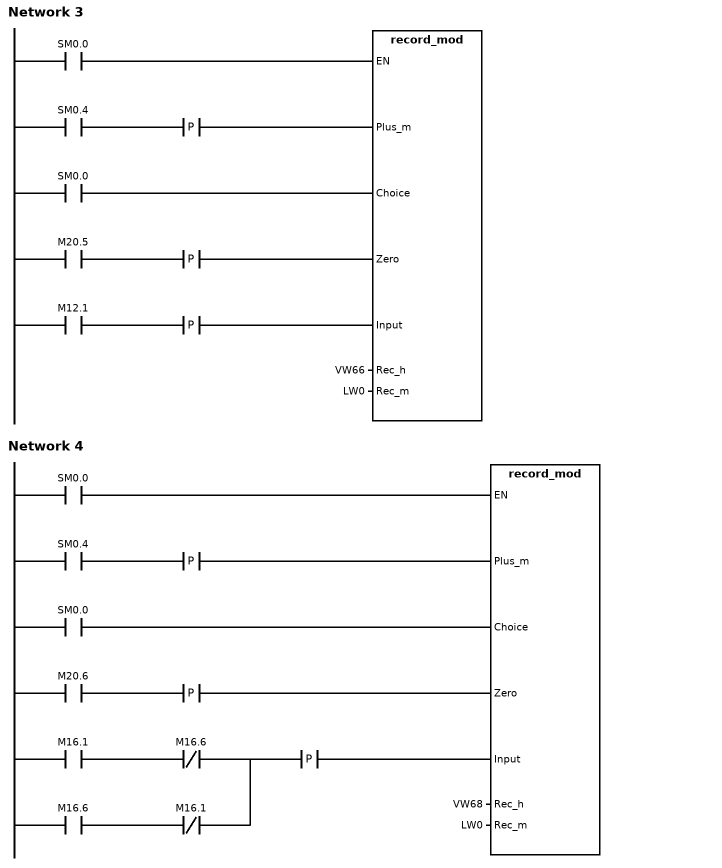
[picture p24: SBR11 networks 3-4]
Network 3
LD     SM0.0
=      L60.0
LD     SM0.4
EU
=      L63.7
LD     SM0.0
=      L63.6
LD     M20.5
EU
=      L63.5
LD     M12.1
EU
=      L63.4
LD     L60.0
CALL   record_mod:SBR13, L63.7, L63.6, L63.5, L63.4, VW66, LW0
Network 4
LD     SM0.0
=      L60.0
LD     SM0.4
EU
=      L63.7
LD     SM0.0
=      L63.6
LD     M20.6
EU
=      L63.5
LD     M16.1
AN     M16.6
LD     M16.6
AN     M16.1
OLD
EU
=      L63.4
LD     L60.0
CALL   record_mod:SBR13, L63.7, L63.6, L63.5, L63.4, VW68, LW0
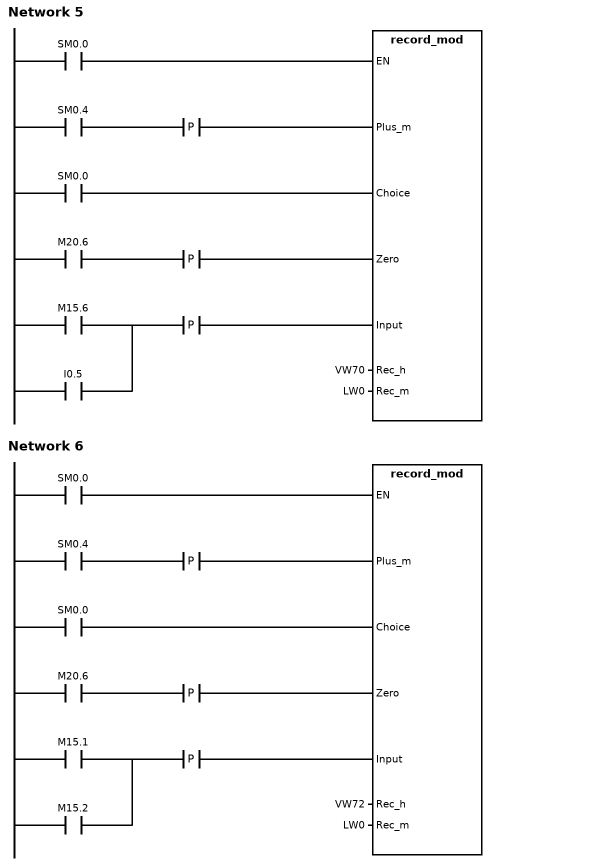
Network 5
LD     SM0.0
=      L60.0
LD     SM0.4
EU
=      L63.7
LD     SM0.0
=      L63.6
LD     M20.6
EU
=      L63.5
LD     M15.6
O      I0.5
EU
=      L63.4
LD     L60.0
CALL   record_mod:SBR13, L63.7, L63.6, L63.5, L63.4, VW70, LW0
Network 6
LD     SM0.0
=      L60.0
LD     SM0.4
EU
=      L63.7
LD     SM0.0
=      L63.6
LD     M20.6
EU
=      L63.5
LD     M15.1
O      M15.2
EU
=      L63.4
LD     L60.0
CALL   record_mod:SBR13, L63.7, L63.6, L63.5, L63.4, VW72, LW0
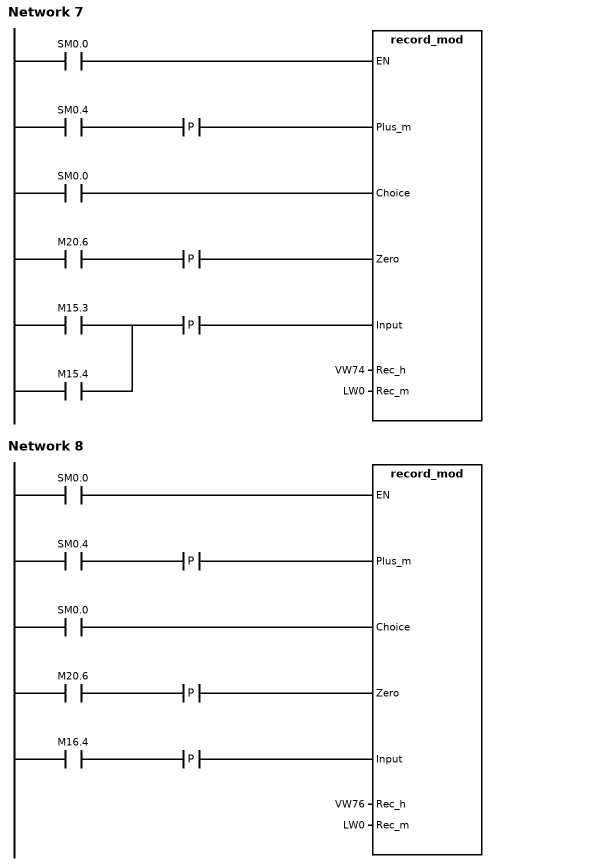
Network 7
LD     SM0.0
=      L60.0
LD     SM0.4
EU
=      L63.7
LD     SM0.0
=      L63.6
LD     M20.6
EU
=      L63.5
LD     M15.3
O      M15.4
EU
=      L63.4
LD     L60.0
CALL   record_mod:SBR13, L63.7, L63.6, L63.5, L63.4, VW74, LW0
Network 8
LD     SM0.0
=      L60.0
LD     SM0.4
EU
=      L63.7
LD     SM0.0
=      L63.6
LD     M20.6
EU
=      L63.5
LD     M16.4
EU
=      L63.4
LD     L60.0
CALL   record_mod:SBR13, L63.7, L63.6, L63.5, L63.4, VW76, LW0
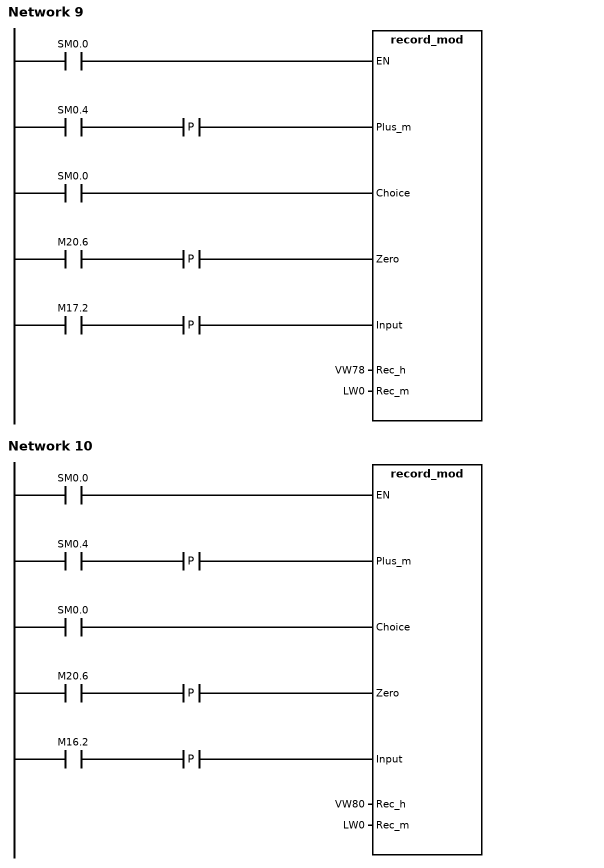
Network 9
LD     SM0.0
=      L60.0
LD     SM0.4
EU
=      L63.7
LD     SM0.0
=      L63.6
LD     M20.6
EU
=      L63.5
LD     M17.2
EU
=      L63.4
LD     L60.0
CALL   record_mod:SBR13, L63.7, L63.6, L63.5, L63.4, VW78, LW0
Network 10
LD     SM0.0
=      L60.0
LD     SM0.4
EU
=      L63.7
LD     SM0.0
=      L63.6
LD     M20.6
EU
=      L63.5
LD     M16.2
EU
=      L63.4
LD     L60.0
CALL   record_mod:SBR13, L63.7, L63.6, L63.5, L63.4, VW80, LW0
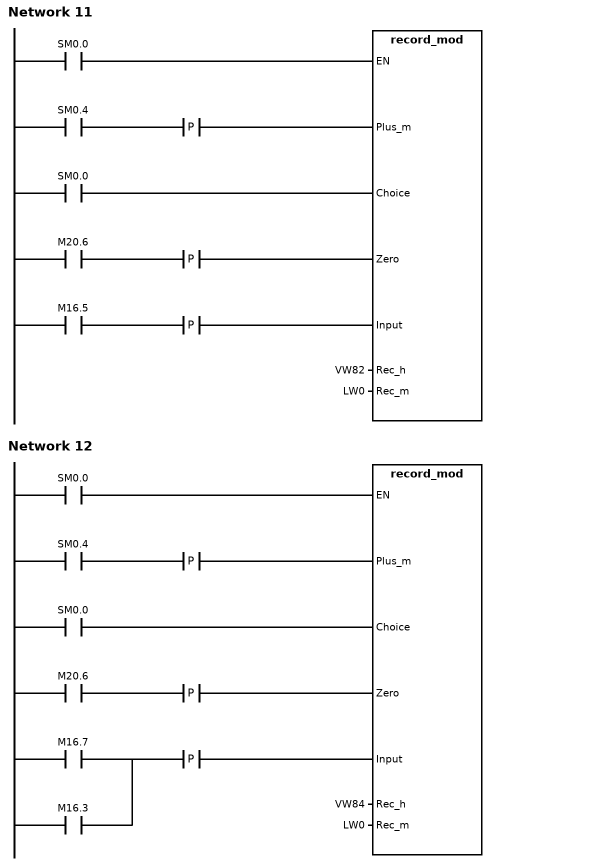
Network 11
LD     SM0.0
=      L60.0
LD     SM0.4
EU
=      L63.7
LD     SM0.0
=      L63.6
LD     M20.6
EU
=      L63.5
LD     M16.5
EU
=      L63.4
LD     L60.0
CALL   record_mod:SBR13, L63.7, L63.6, L63.5, L63.4, VW82, LW0
Network 12
LD     SM0.0
=      L60.0
LD     SM0.4
EU
=      L63.7
LD     SM0.0
=      L63.6
LD     M20.6
EU
=      L63.5
LD     M16.7
O      M16.3
EU
=      L63.4
LD     L60.0
CALL   record_mod:SBR13, L63.7, L63.6, L63.5, L63.4, VW84, LW0
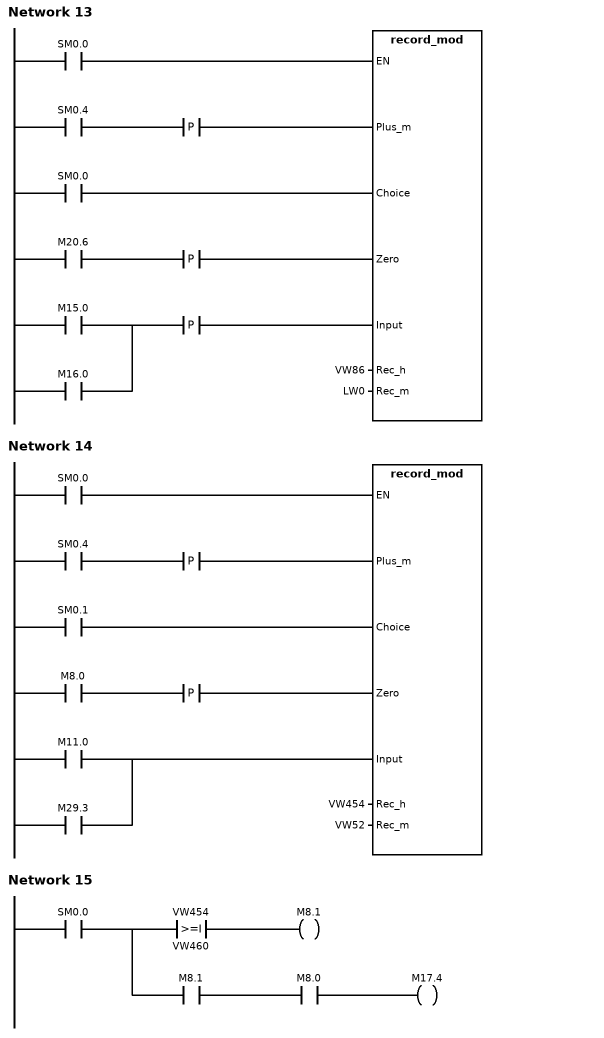
Network 13
LD     SM0.0
=      L60.0
LD     SM0.4
EU
=      L63.7
LD     SM0.0
=      L63.6
LD     M20.6
EU
=      L63.5
LD     M15.0
O      M16.0
EU
=      L63.4
LD     L60.0
CALL   record_mod:SBR13, L63.7, L63.6, L63.5, L63.4, VW86, LW0
Network 14
LD     SM0.0
=      L60.0
LD     SM0.4
EU
=      L63.7
LD     SM0.1
=      L63.6
LD     M8.0
EU
=      L63.5
LD     M11.0
O      M29.3
=      L63.4
LD     L60.0
CALL   record_mod:SBR13, L63.7, L63.6, L63.5, L63.4, VW454, VW52
Network 15
LD     SM0.0
LPS
AW>=   VW454, VW460
=      M8.1
LPP
A      M8.1
A      M8.0
=      M17.4
END_SUBROUTINE_BLOCK

// SBR12: protected block, not included

SUBROUTINE_BLOCK record_mod:SBR13
TITLE=
VAR_INPUT
Plus_m:BOOL;	// L0.0 
Choice:BOOL;	// L0.1 
Zero:BOOL;	// L0.2 
Input:BOOL;	// L0.3 
END_VAR
VAR_IN_OUT
Rec_h:WORD;	// LW1 
Rec_m:WORD;	// LW3 
END_VAR
BEGIN
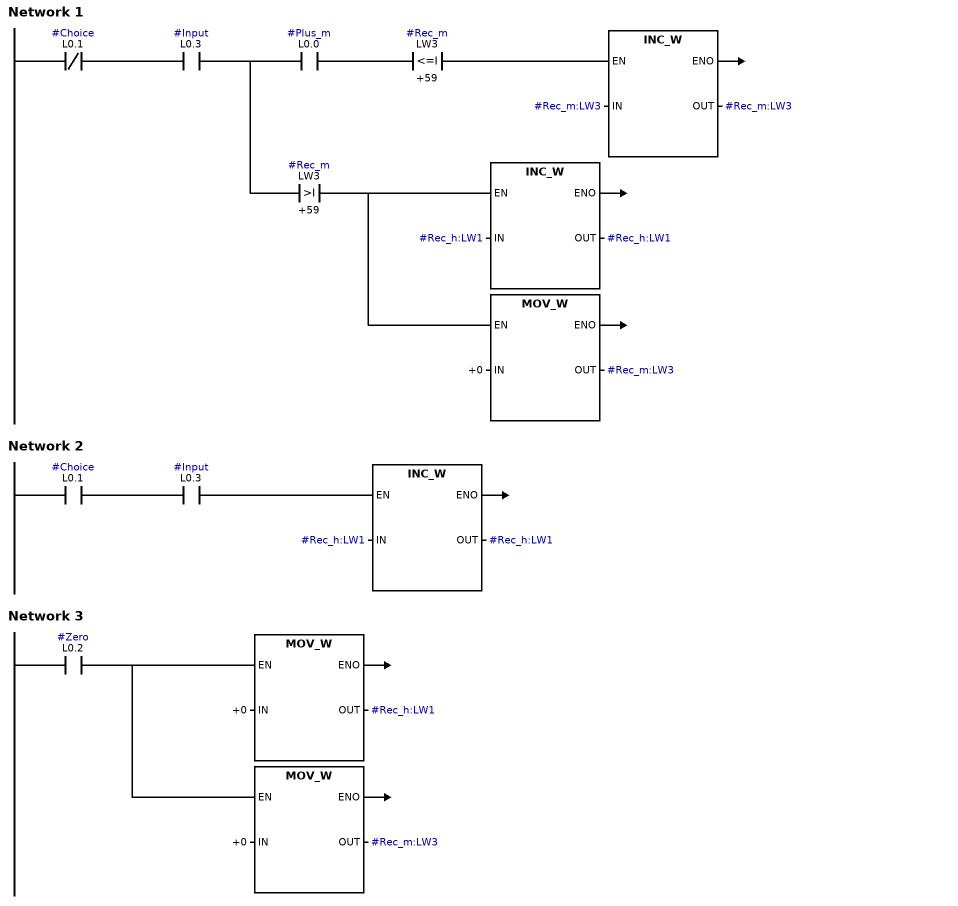
Network 1
LDN    #Choice:L0.1
A      #Input:L0.3
LPS
A      #Plus_m:L0.0
AW<=   #Rec_m:LW3, +59
INCW   #Rec_m:LW3
LPP
AW>    #Rec_m:LW3, +59
INCW   #Rec_h:LW1
MOVW   +0, #Rec_m:LW3
Network 2
LD     #Choice:L0.1
A      #Input:L0.3
INCW   #Rec_h:LW1
Network 3
LD     #Zero:L0.2
MOVW   +0, #Rec_h:LW1
MOVW   +0, #Rec_m:LW3
END_SUBROUTINE_BLOCK

SUBROUTINE_BLOCK Burner:SBR14
TITLE=
BEGIN
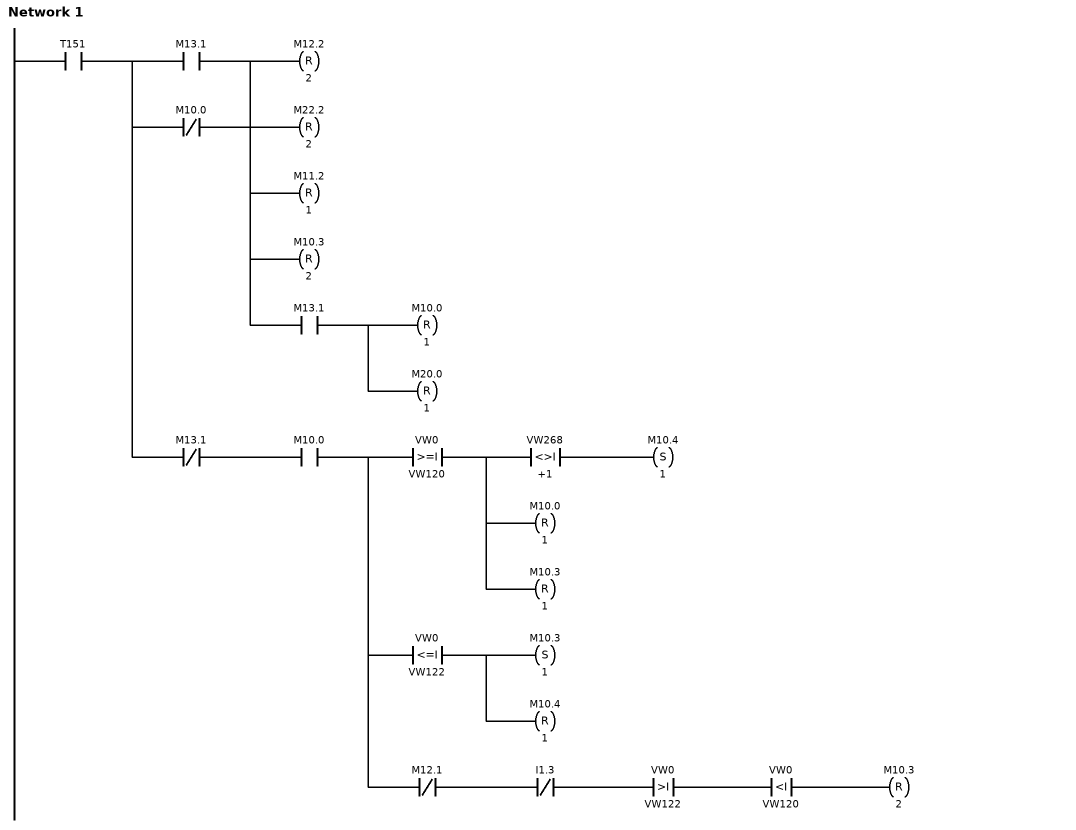
Network 1
LD     T151
LPS
LD     M13.1
ON     M10.0
ALD
R      M12.2, 2
R      M22.2, 2
R      M11.2, 1
R      M10.3, 2
A      M13.1
R      M10.0, 1
R      M20.0, 1
LPP
AN     M13.1
A      M10.0
LPS
AW>=   VW0, VW120
LPS
AW<>   VW268, +1
S      M10.4, 1
LRD
R      M10.0, 1
LPP
R      M10.3, 1
LRD
AW<=   VW0, VW122
S      M10.3, 1
R      M10.4, 1
LPP
AN     M12.1
AN     I1.3
AW>    VW0, VW122
AW<    VW0, VW120
R      M10.3, 2
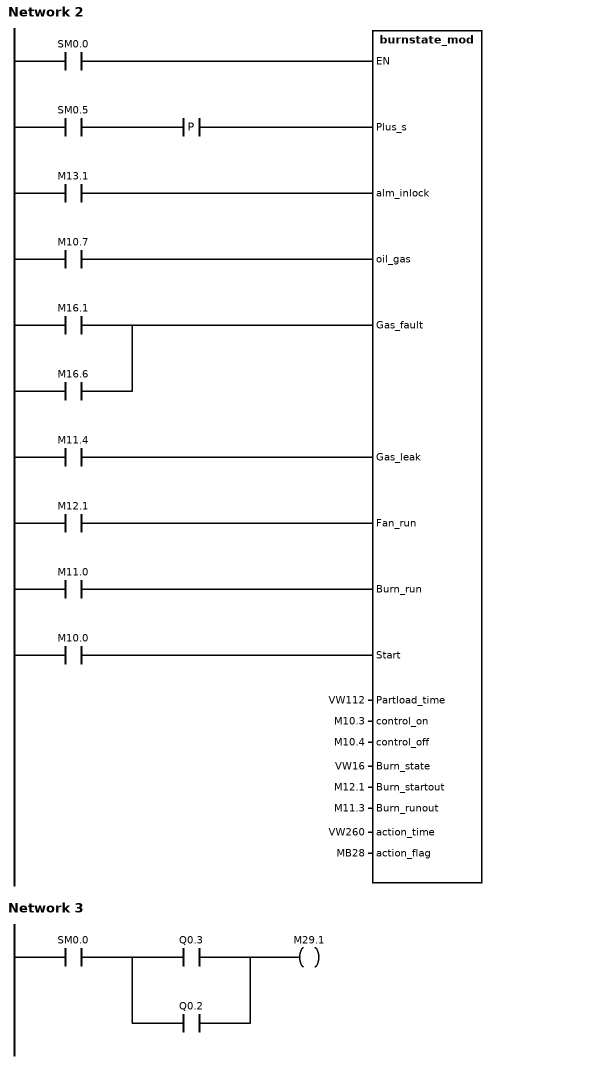
Network 2
LD     SM0.0
=      L60.0
LD     SM0.5
EU
=      L63.7
LD     M13.1
=      L63.6
LD     M10.7
=      L63.5
LD     M16.1
O      M16.6
=      L63.4
LD     M11.4
=      L63.3
LD     M12.1
=      L63.2
LD     M11.0
=      L63.1
LD     M10.0
=      L63.0
LD     L60.0
CALL   burnstate_mod:SBR23, L63.7, L63.6, L63.5, L63.4, L63.3, L63.2, L63.1, L63.0, VW112, M10.3, M10.4, VW16, M12.1, M11.3, VW260, MB28
Network 3
LD     SM0.0
LD     Q0.3
O      Q0.2
ALD
=      M29.1
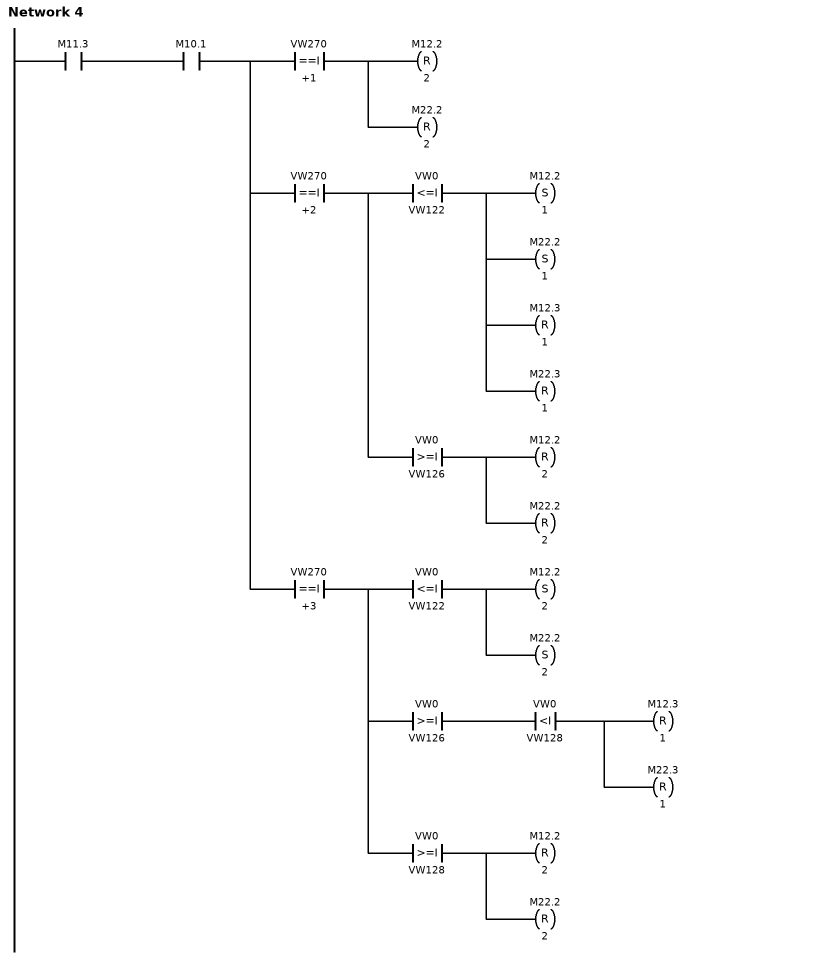
Network 4
LD     M11.3
A      M10.1
LPS
AW=    VW270, +1
R      M12.2, 2
R      M22.2, 2
LRD
AW=    VW270, +2
LPS
AW<=   VW0, VW122
S      M12.2, 1
S      M22.2, 1
R      M12.3, 1
R      M22.3, 1
LPP
AW>=   VW0, VW126
R      M12.2, 2
R      M22.2, 2
LPP
AW=    VW270, +3
LPS
AW<=   VW0, VW122
S      M12.2, 2
S      M22.2, 2
LRD
AW>=   VW0, VW126
AW<    VW0, VW128
R      M12.3, 1
R      M22.3, 1
LPP
AW>=   VW0, VW128
R      M12.2, 2
R      M22.2, 2
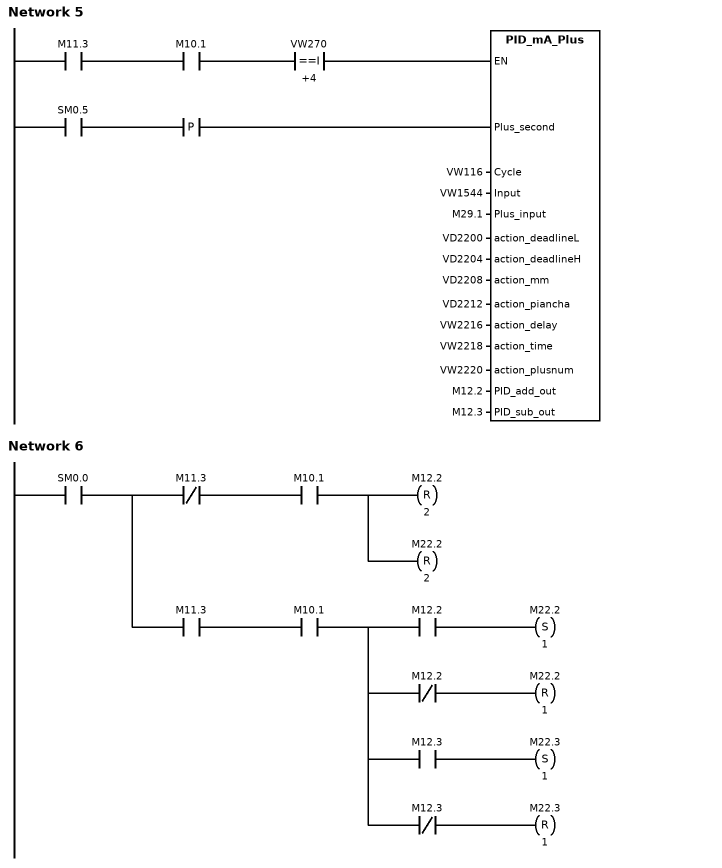
Network 5
LD     M11.3
A      M10.1
AW=    VW270, +4
=      L60.0
LD     SM0.5
EU
=      L63.7
LD     L60.0
CALL   PID_mA_Plus:SBR16, L63.7, VW116, VW1544, M29.1, VD2200, VD2204, VD2208, VD2212, VW2216, VW2218, VW2220, M12.2, M12.3
Network 6
LD     SM0.0
LPS
AN     M11.3
A      M10.1
R      M12.2, 2
R      M22.2, 2
LPP
A      M11.3
A      M10.1
LPS
A      M12.2
S      M22.2, 1
LRD
AN     M12.2
R      M22.2, 1
LRD
A      M12.3
S      M22.3, 1
LPP
AN     M12.3
R      M22.3, 1
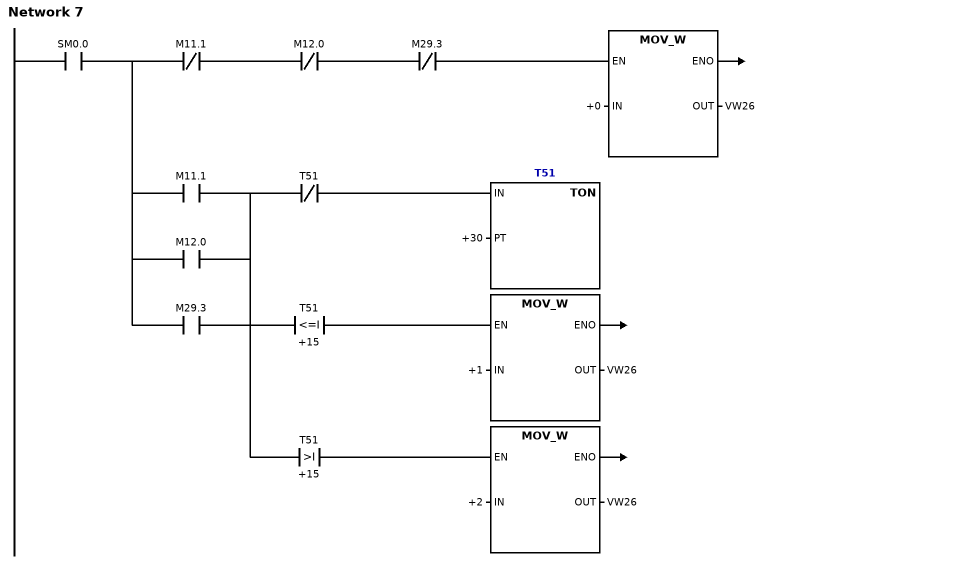
Network 7
LD     SM0.0
LPS
AN     M11.1
AN     M12.0
AN     M29.3
MOVW   +0, VW26
LPP
LD     M11.1
O      M12.0
O      M29.3
ALD
LPS
AN     T51
TON    T51, +30
LRD
AW<=   T51, +15
MOVW   +1, VW26
LPP
AW>    T51, +15
MOVW   +2, VW26
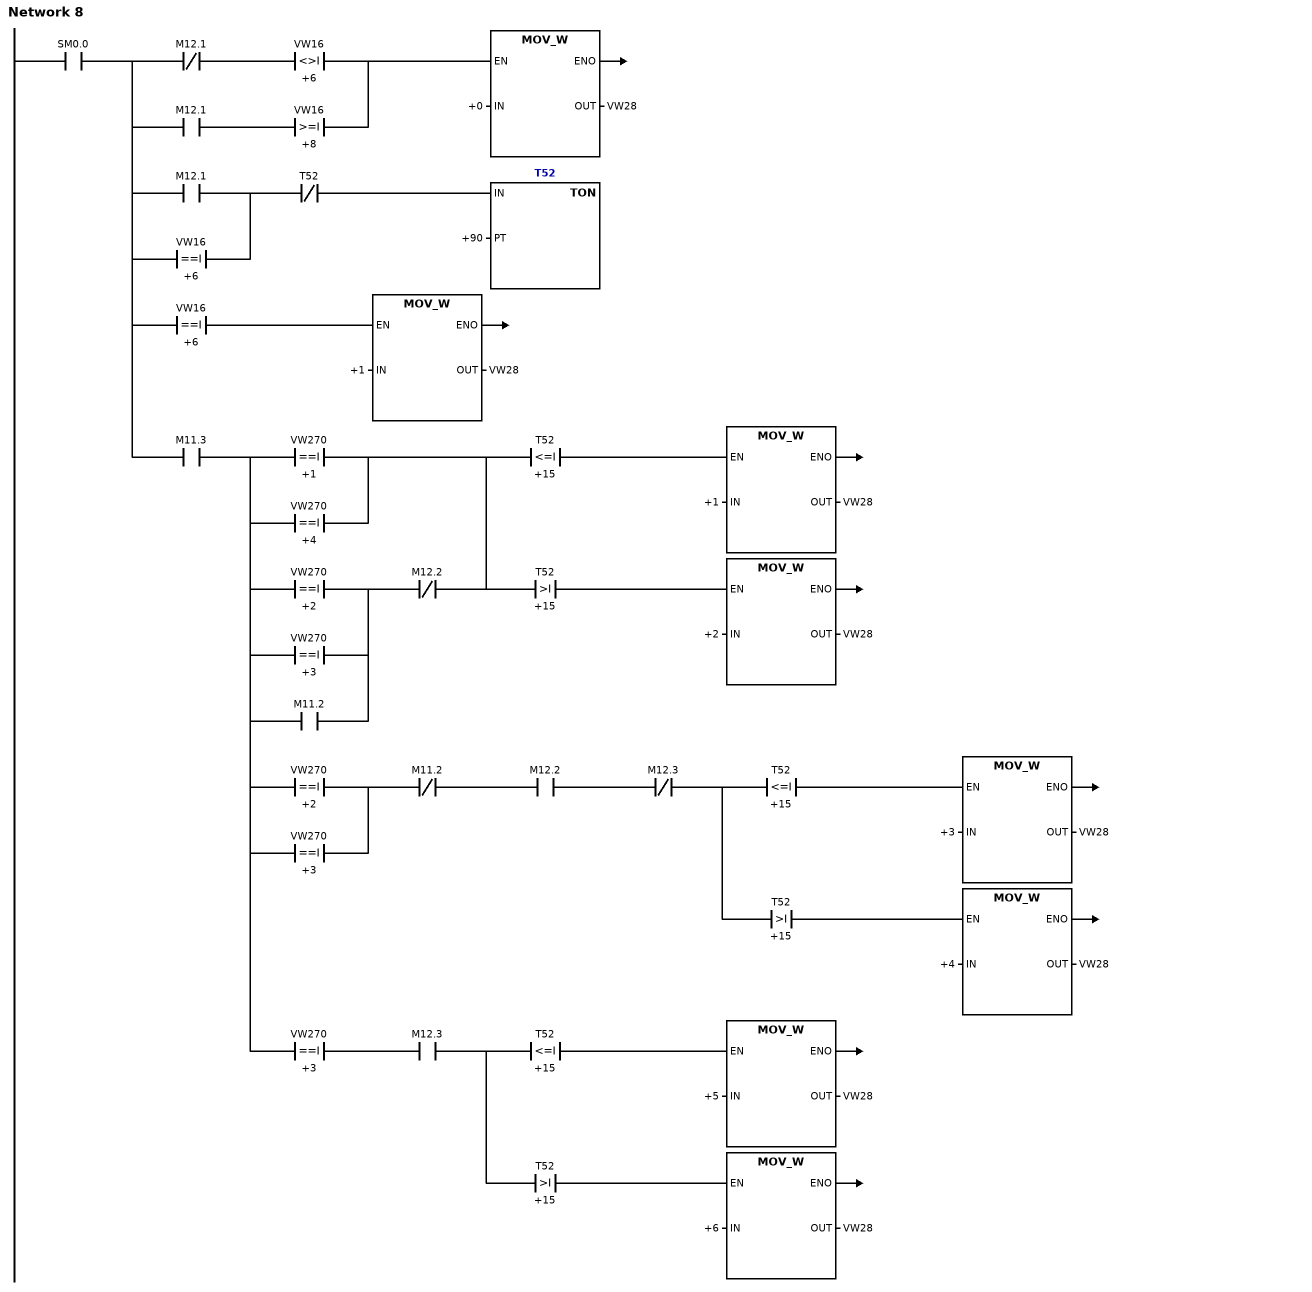
Network 8
LD     SM0.0
LPS
LDN    M12.1
AW<>   VW16, +6
LD     M12.1
AW>=   VW16, +8
OLD
ALD
MOVW   +0, VW28
LRD
LD     M12.1
OW=    VW16, +6
ALD
AN     T52
TON    T52, +90
LRD
AW=    VW16, +6
MOVW   +1, VW28
LPP
A      M11.3
LPS
LDW=   VW270, +1
OW=    VW270, +4
LDW=   VW270, +2
OW=    VW270, +3
O      M11.2
AN     M12.2
OLD
ALD
LPS
AW<=   T52, +15
MOVW   +1, VW28
LPP
AW>    T52, +15
MOVW   +2, VW28
LPP
LPS
LDW=   VW270, +2
OW=    VW270, +3
AN     M11.2
A      M12.2
AN     M12.3
ALD
LPS
AW<=   T52, +15
MOVW   +3, VW28
LPP
AW>    T52, +15
MOVW   +4, VW28
LPP
AW=    VW270, +3
A      M12.3
LPS
AW<=   T52, +15
MOVW   +5, VW28
LPP
AW>    T52, +15
MOVW   +6, VW28
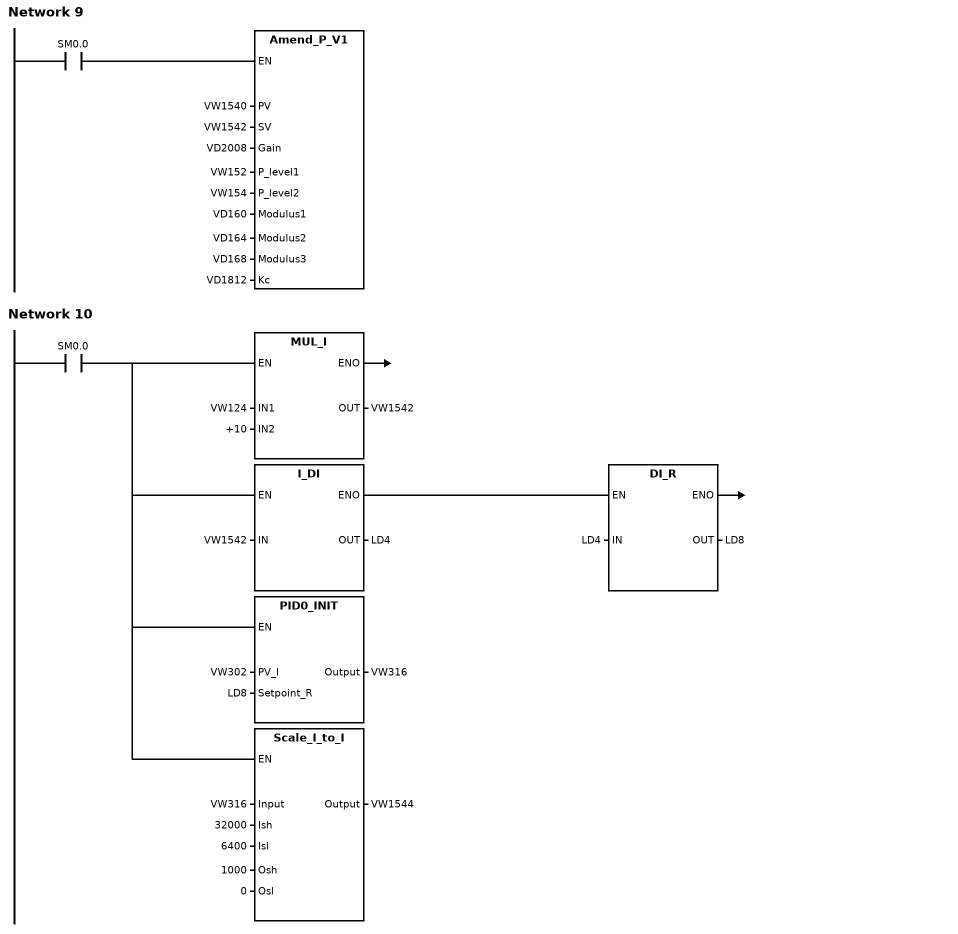
Network 9
LD     SM0.0
CALL   Amend_P_V1:SBR33, VW1540, VW1542, VD2008, VW152, VW154, VD160, VD164, VD168, VD1812
Network 10
LD     SM0.0
LPS
MOVW   VW124, VW1542
*I     +10, VW1542
ITD    VW1542, LD4
AENO
DTR    LD4, LD8
LRD
CALL   PID0_INIT:SBR6, VW302, LD8, VW316
LPP
CALL   Scale_I_to_I:SBR3, VW316, 32000, 6400, 1000, 0, VW1544
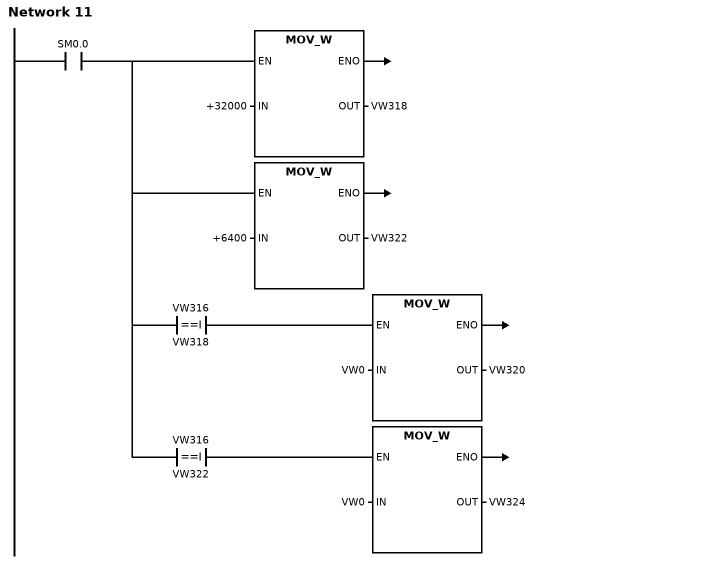
Network 11
LD     SM0.0
LPS
MOVW   +32000, VW318
MOVW   +6400, VW322
AW=    VW316, VW318
MOVW   VW0, VW320
LPP
AW=    VW316, VW322
MOVW   VW0, VW324
END_SUBROUTINE_BLOCK

SUBROUTINE_BLOCK Invter_Con:SBR15
TITLE=
BEGIN
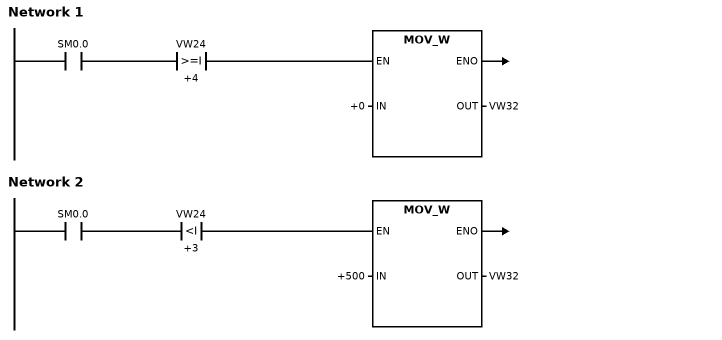
Network 1
LD     SM0.0
AW>=   VW24, +4
MOVW   +0, VW32
Network 2
LD     SM0.0
AW<    VW24, +3
MOVW   +500, VW32
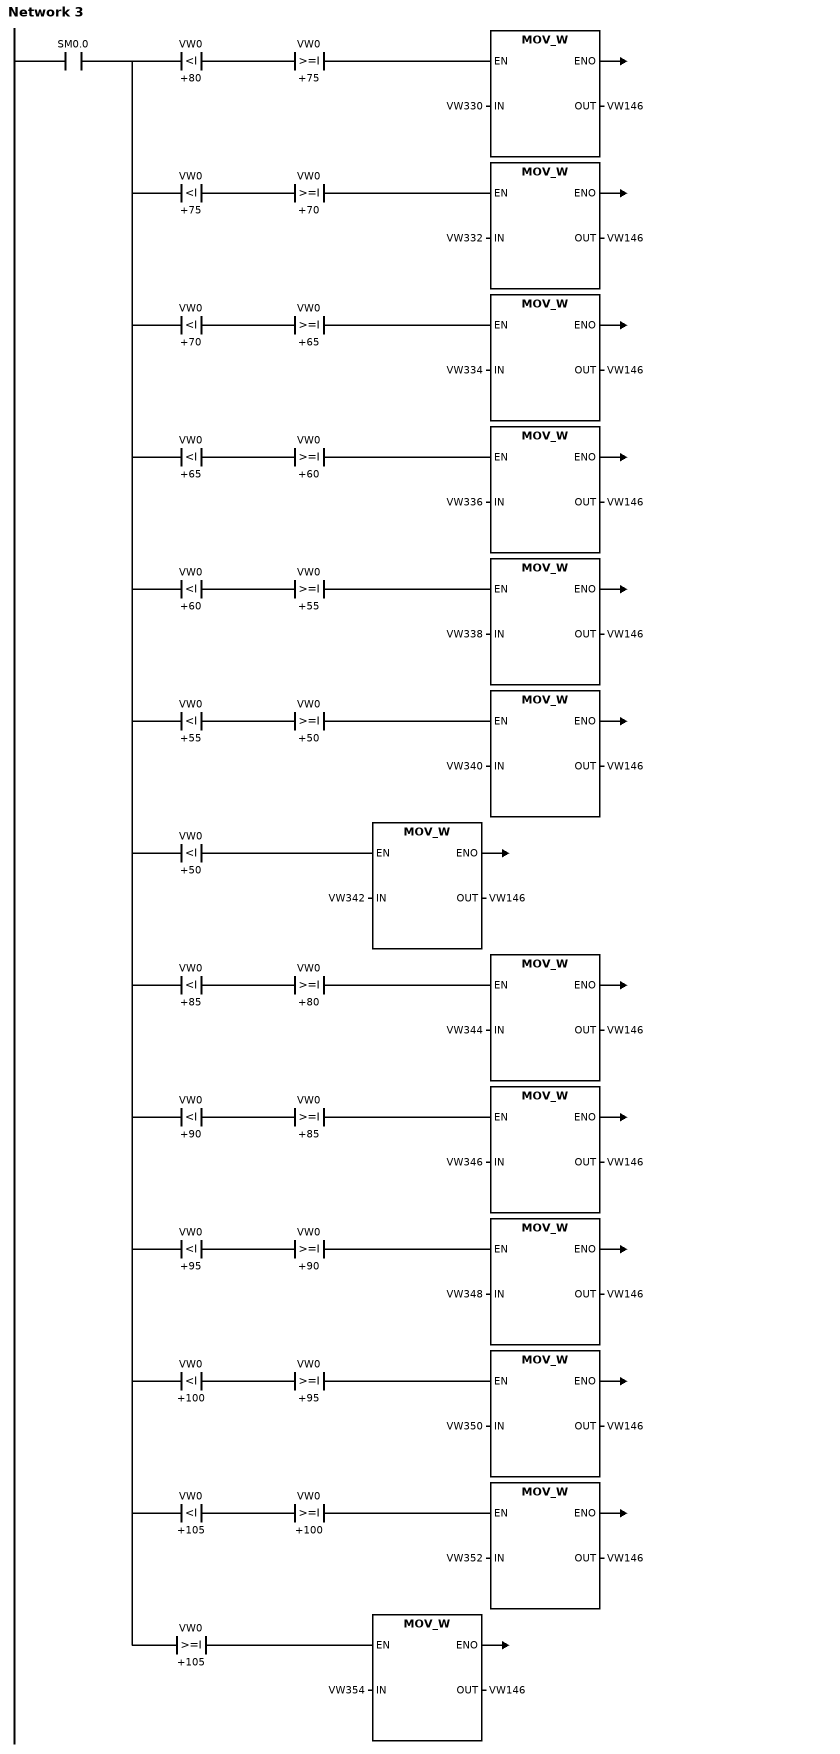
Network 3
LD     SM0.0
LPS
AW<    VW0, +80
AW>=   VW0, +75
MOVW   VW330, VW146
LRD
AW<    VW0, +75
AW>=   VW0, +70
MOVW   VW332, VW146
LRD
AW<    VW0, +70
AW>=   VW0, +65
MOVW   VW334, VW146
LRD
AW<    VW0, +65
AW>=   VW0, +60
MOVW   VW336, VW146
LRD
AW<    VW0, +60
AW>=   VW0, +55
MOVW   VW338, VW146
LRD
AW<    VW0, +55
AW>=   VW0, +50
MOVW   VW340, VW146
LRD
AW<    VW0, +50
MOVW   VW342, VW146
LRD
AW<    VW0, +85
AW>=   VW0, +80
MOVW   VW344, VW146
LRD
AW<    VW0, +90
AW>=   VW0, +85
MOVW   VW346, VW146
LRD
AW<    VW0, +95
AW>=   VW0, +90
MOVW   VW348, VW146
LRD
AW<    VW0, +100
AW>=   VW0, +95
MOVW   VW350, VW146
LRD
AW<    VW0, +105
AW>=   VW0, +100
MOVW   VW352, VW146
LPP
AW>=   VW0, +105
MOVW   VW354, VW146
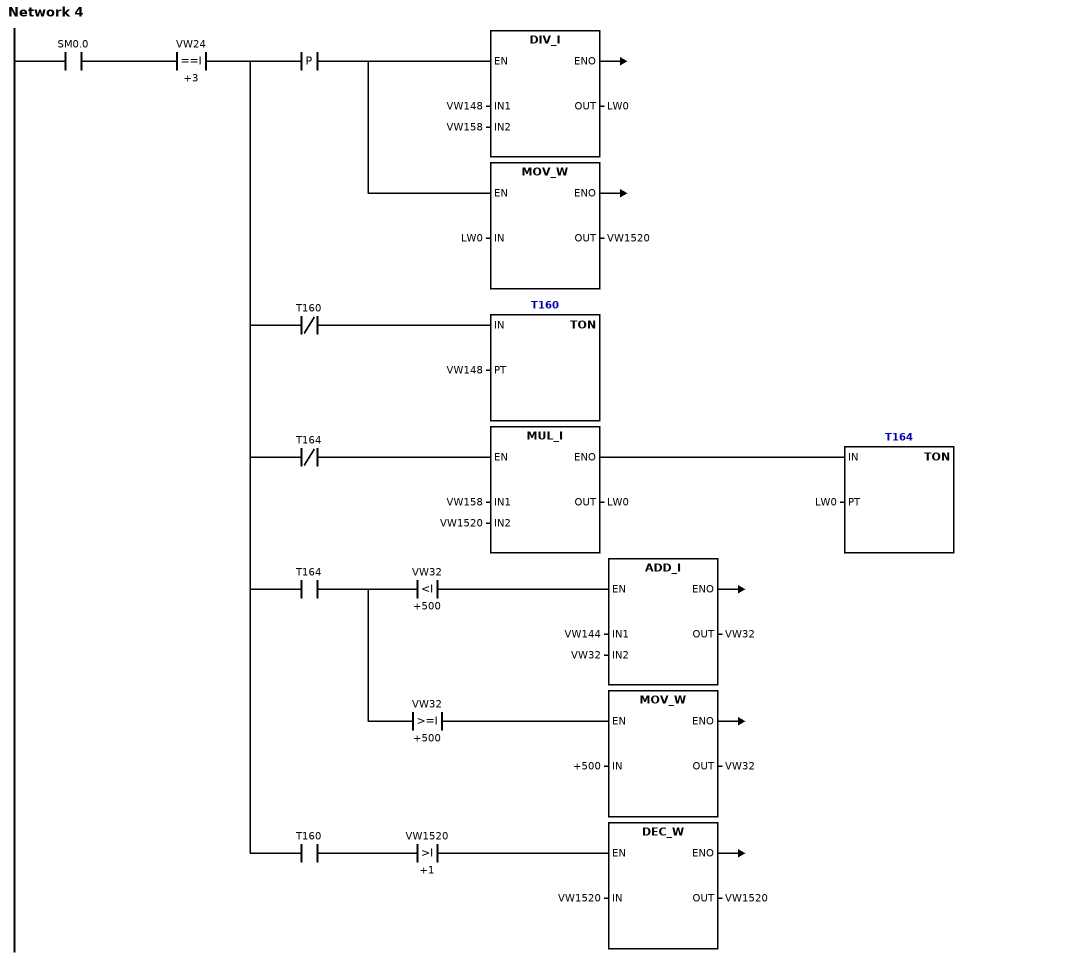
Network 4
LD     SM0.0
AW=    VW24, +3
LPS
EU
MOVW   VW148, LW0
/I     VW158, LW0
MOVW   LW0, VW1520
LRD
LPS
AN     T160
TON    T160, VW148
LPP
AN     T164
MOVW   VW158, LW0
AENO
*I     VW1520, LW0
AENO
TON    T164, LW0
LRD
A      T164
LPS
AW<    VW32, +500
+I     VW144, VW32
LPP
AW>=   VW32, +500
MOVW   +500, VW32
LPP
A      T160
AW>    VW1520, +1
DECW   VW1520
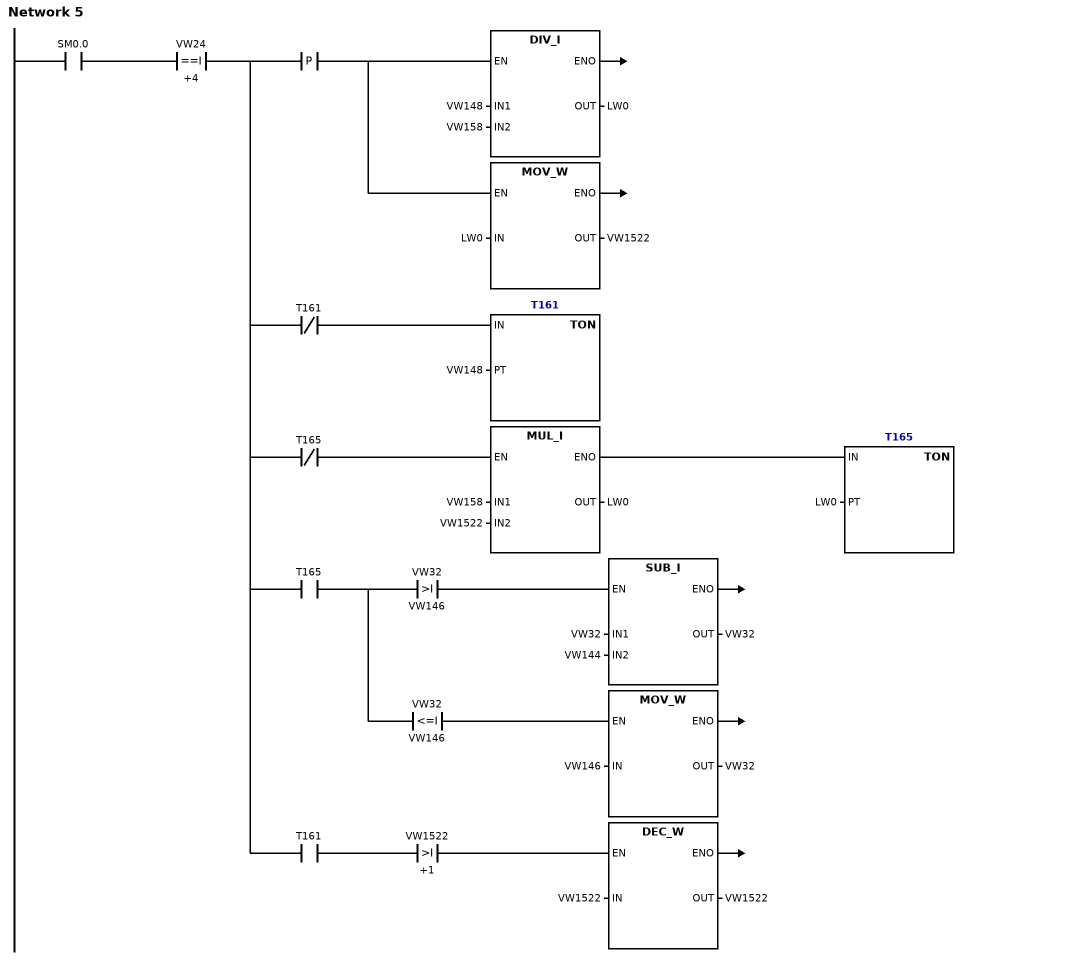
Network 5
LD     SM0.0
AW=    VW24, +4
LPS
EU
MOVW   VW148, LW0
/I     VW158, LW0
MOVW   LW0, VW1522
LRD
LPS
AN     T161
TON    T161, VW148
LPP
AN     T165
MOVW   VW158, LW0
AENO
*I     VW1522, LW0
AENO
TON    T165, LW0
LRD
A      T165
LPS
AW>    VW32, VW146
-I     VW144, VW32
LPP
AW<=   VW32, VW146
MOVW   VW146, VW32
LPP
A      T161
AW>    VW1522, +1
DECW   VW1522
END_SUBROUTINE_BLOCK

// SBR16: protected block, not included

SUBROUTINE_BLOCK Digtal_In:SBR17
TITLE=
BEGIN
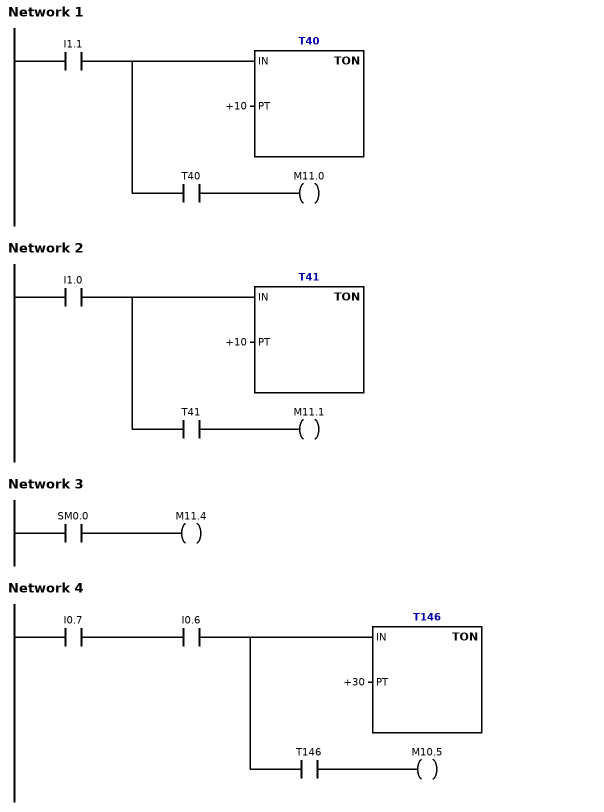
Network 1
LD     I1.1
TON    T40, +10
A      T40
=      M11.0
Network 2
LD     I1.0
TON    T41, +10
A      T41
=      M11.1
Network 3
LD     SM0.0
=      M11.4
Network 4
LD     I0.7
A      I0.6
TON    T146, +30
A      T146
=      M10.5
END_SUBROUTINE_BLOCK

SUBROUTINE_BLOCK Read_Rtc:SBR18
TITLE=
VAR_IN_OUT
R_Time_Y:WORD;	// LW0 
R_Time_M:WORD;	// LW2 
R_Time_D:WORD;	// LW4 
R_Time_H:WORD;	// LW6 
R_Time_m:WORD;	// LW8 
R_Time_S:WORD;	// LW10 
R_Time_W:WORD;	// LW12 
END_VAR
BEGIN
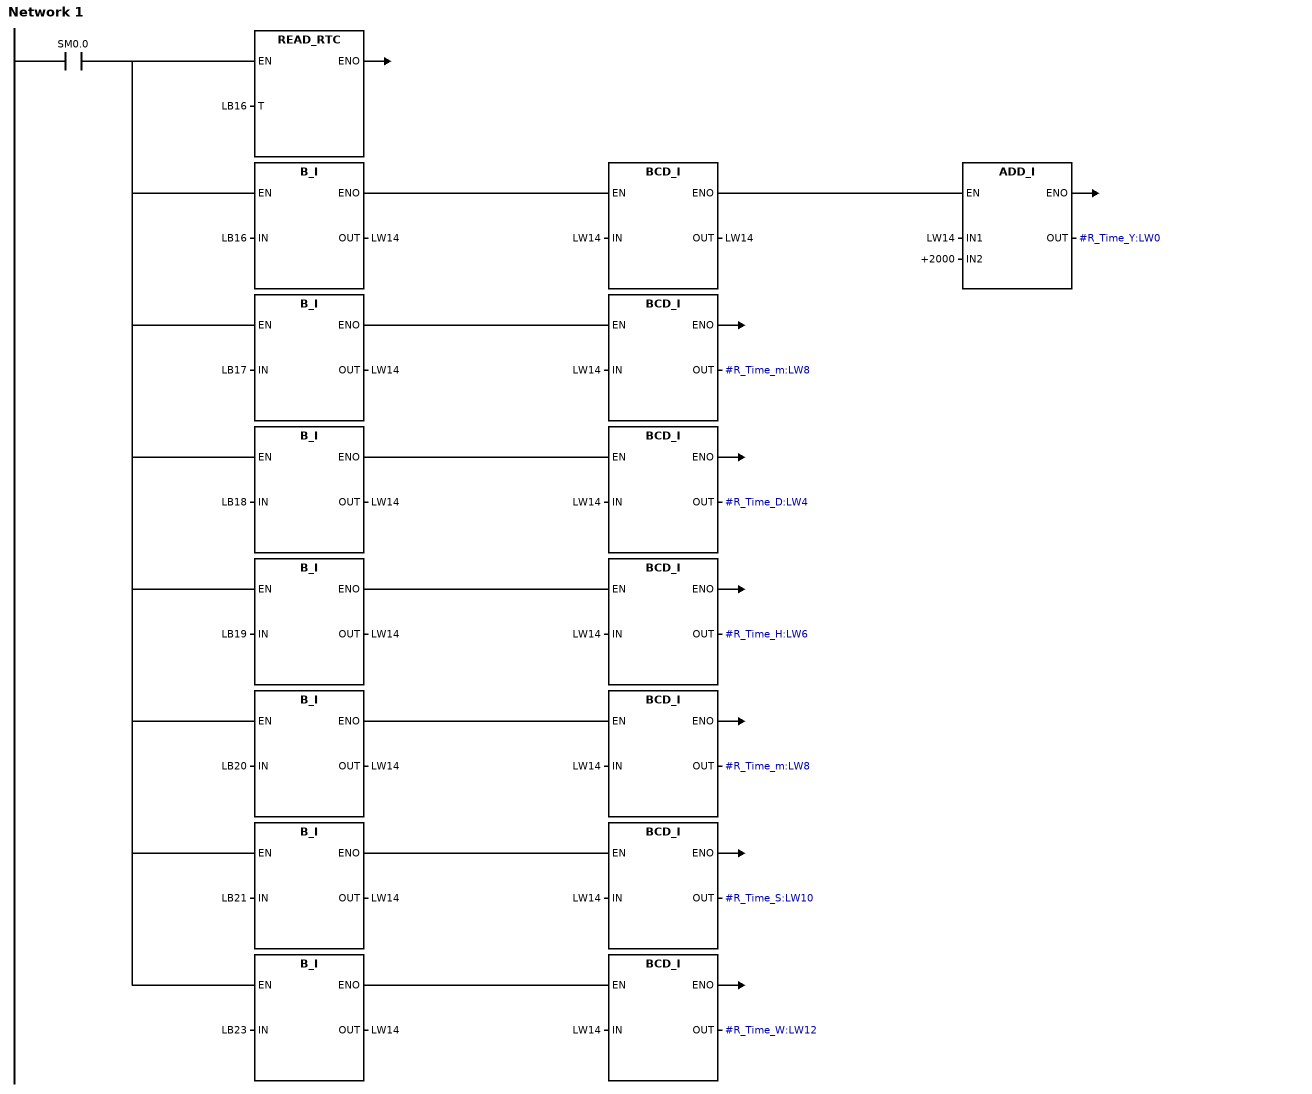
Network 1
LD     SM0.0
LPS
TODR   LB16
BTI    LB16, LW14
AENO
BCDI   LW14
AENO
MOVW   LW14, #R_Time_Y:LW0
+I     +2000, #R_Time_Y:LW0
LRD
BTI    LB17, LW14
AENO
MOVW   LW14, #R_Time_M:LW2
BCDI   #R_Time_M:LW2
LRD
BTI    LB18, LW14
AENO
MOVW   LW14, #R_Time_D:LW4
BCDI   #R_Time_D:LW4
LRD
BTI    LB19, LW14
AENO
MOVW   LW14, #R_Time_H:LW6
BCDI   #R_Time_H:LW6
LRD
BTI    LB20, LW14
AENO
MOVW   LW14, #R_Time_m:LW8
BCDI   #R_Time_m:LW8
LRD
BTI    LB21, LW14
AENO
MOVW   LW14, #R_Time_S:LW10
BCDI   #R_Time_S:LW10
LPP
BTI    LB23, LW14
AENO
MOVW   LW14, #R_Time_W:LW12
BCDI   #R_Time_W:LW12
END_SUBROUTINE_BLOCK

SUBROUTINE_BLOCK RealTime:SBR19
TITLE=
BEGIN
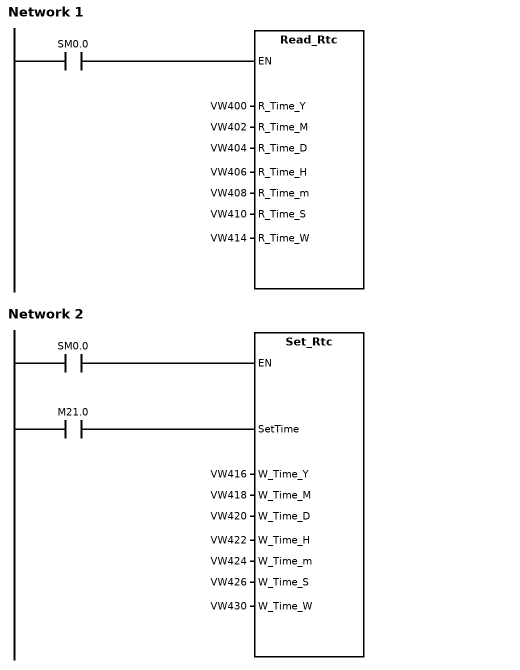
Network 1
LD     SM0.0
CALL   Read_Rtc:SBR18, VW400, VW402, VW404, VW406, VW408, VW410, VW414
Network 2
LD     SM0.0
=      L60.0
LD     M21.0
=      L63.7
LD     L60.0
CALL   Set_Rtc:SBR20, L63.7, VW416, VW418, VW420, VW422, VW424, VW426, VW430
END_SUBROUTINE_BLOCK

SUBROUTINE_BLOCK Set_Rtc:SBR20
TITLE=
VAR_INPUT
SetTime:BOOL;	// L0.0 
END_VAR
VAR_IN_OUT
W_Time_Y:WORD;	// LW1 
W_Time_M:WORD;	// LW3 
W_Time_D:WORD;	// LW5 
W_Time_H:WORD;	// LW7 
W_Time_m:WORD;	// LW9 
W_Time_S:WORD;	// LW11 
W_Time_W:WORD;	// LW13 
END_VAR
BEGIN
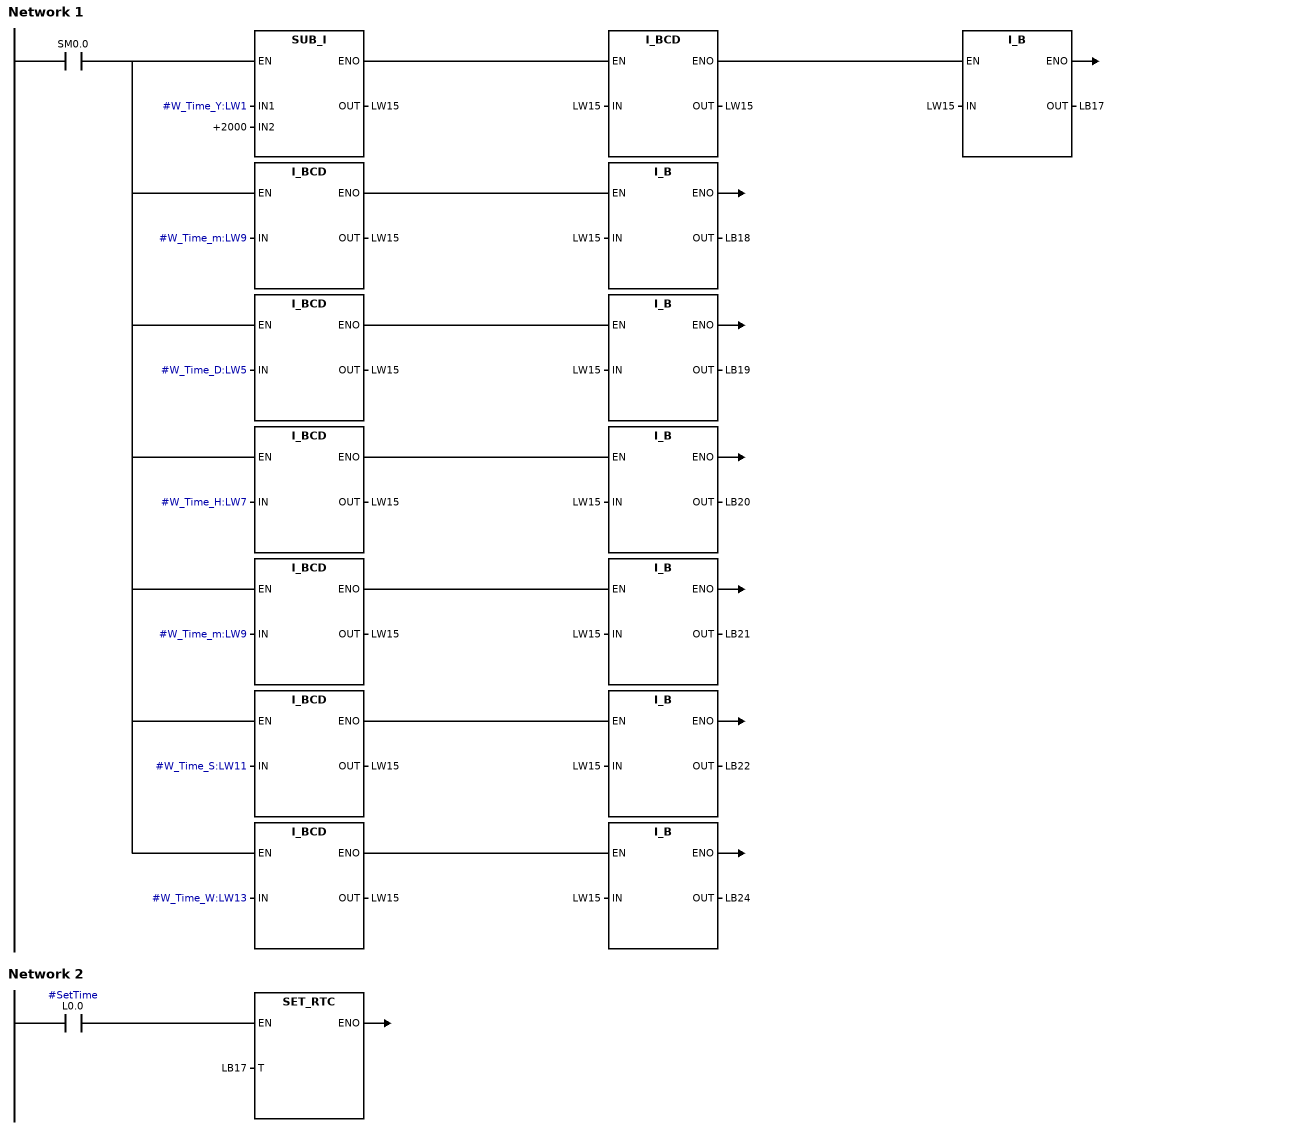
Network 1
LD     SM0.0
LPS
MOVW   #W_Time_Y:LW1, LW15
AENO
-I     +2000, LW15
AENO
IBCD   LW15
AENO
ITB    LW15, LB17
LRD
MOVW   #W_Time_M:LW3, LW15
AENO
IBCD   LW15
AENO
ITB    LW15, LB18
LRD
MOVW   #W_Time_D:LW5, LW15
AENO
IBCD   LW15
AENO
ITB    LW15, LB19
LRD
MOVW   #W_Time_H:LW7, LW15
AENO
IBCD   LW15
AENO
ITB    LW15, LB20
LRD
MOVW   #W_Time_m:LW9, LW15
AENO
IBCD   LW15
AENO
ITB    LW15, LB21
LRD
MOVW   #W_Time_S:LW11, LW15
AENO
IBCD   LW15
AENO
ITB    LW15, LB22
LPP
MOVW   #W_Time_W:LW13, LW15
AENO
IBCD   LW15
AENO
ITB    LW15, LB24
Network 2
LD     #SetTime:L0.0
TODW   LB17
END_SUBROUTINE_BLOCK

// SBR23: protected block, not included

SUBROUTINE_BLOCK Output:SBR24
TITLE=
BEGIN
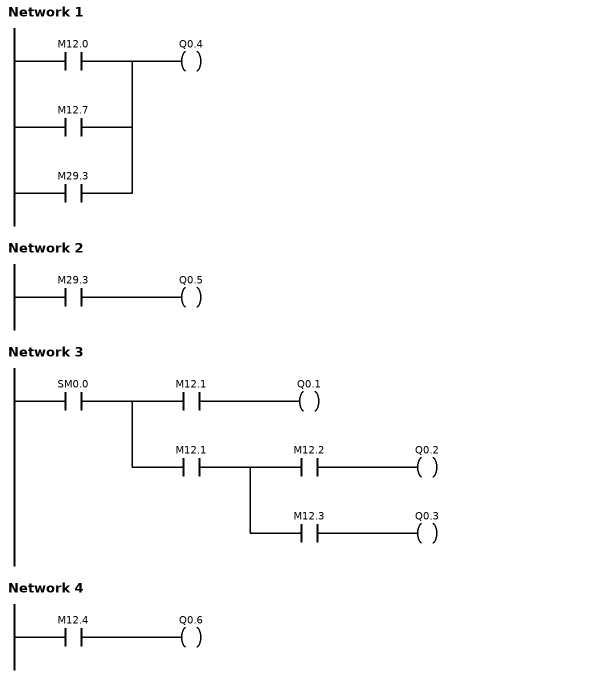
Network 1
LD     M12.0
O      M12.7
O      M29.3
=      Q0.4
Network 2
LD     M29.3
=      Q0.5
Network 3
LD     SM0.0
LPS
A      M12.1
=      Q0.1
LPP
A      M12.1
LPS
A      M12.2
=      Q0.2
LPP
A      M12.3
=      Q0.3
Network 4
LD     M12.4
=      Q0.6
